FUNCTION_BLOCK fb_DBSRVInsertRecord
VAR_INPUT
	InsertData:ST_InsertData;
	table:STRING(50);
	DBID:UINT;
	bExecute:bool;
	
END_VAR
VAR_OUTPUT
	bError:BOOL:=FALSE;
	bReady:BOOL:=FALSE;
	
END_VAR
VAR
	nstep:INT:=10;
	sCmd:STRING(255);
	SQLcommand: FB_SQLCommandEvt(sNetid:='',tTimeout:=T#5S);
	Connectdb: FB_sqldatabaseevt(SNetID:='', tTimeout:=T#5S);
	connected:BOOL:=FALSE;
	
END_VAR

IF bExecute THEN
CASE nstep OF 
	10:
			sCmd:=concat('insert into ',table);
			sCmd:=concat(sCmd,  ' (Dátum , temp_set, temp_act, hum_set, hum_act ) values ('); //{Datum},{temp_set},{temp_act},{hum_set}, {hum_act})');
			sCmd:=concat(sCmd,insertdata.Datum);
			sCmd:=concat(sCmd,', ');
			sCmd:=concat(sCmd,insertdata.temp_set);
			sCmd:=concat(sCmd,', ');
			sCmd:=concat(sCmd,insertdata.temp_act);
			sCmd:=concat(sCmd,', ');
			sCmd:=concat(sCmd, insertdata.hum_set);
			sCmd:=concat(sCmd,', ');
			sCmd:=concat(sCmd,insertdata.hum_act);
			sCmd:=concat(sCmd,')');
			nstep:=20;
	20:
			IF connectDB.Connect(DBID) THEN
				IF connectdb.bError THEN
					bError:=TRUE;
				ELSE
					connected:=TRUE;	
				END_IF
			END_IF
			IF connected AND NOT connectDB.bBusy THEN 
				IF connectDB.CreateCmd(pSQLCommand:= ADR(SQLcommand)) THEN
					nstep:=30;
				END_IF
			END_IF		
	30:
		IF SQLcommand.Execute(pSQLCmd:=ADR(sCmd),
							cbSQLCmd:=SIZEOF(sCmd))
			THEN
			IF sqlcommand.bError THEN
				Berror:=TRUE;
			ELSE
			IF NOT SQLcommand.bBusy THEN
				nstep:=40;
			END_IF
			END_IF
		END_IF
	40:	
		IF connectDB.Disconnect() THEN
			IF connectdb.bError THEN
				bError:=TRUE;
			ELSE
				connected:=FALSE;
				bReady:=TRUE;
				bExecute:=FALSE;	
		END_IF
		END_IF		
		
END_CASE
END_IF

METHOD Reset : BOOL
VAR_INPUT
END_VAR
bReady:=FALSE;
nstep:=10;
END_METHOD

END_FUNCTION_BLOCK

(* stored: Version 1.1.0.1, ProductVersion 3.1.4024.2
   POU fb_DBSRVInsertRecord: Id {e335c143-6fa9-41ef-b8f7-d4a9881b27fa}, SpecialFunc None
   Method Reset: Id {b397fd6f-6838-45b1-929d-41d053163da2} *)
